(*
A circular queue implementation for managing `I_Arg`.  
*)
INTERFACE I_ArgQueue EXTENDS I_Debug

(*
Returns the current head index of the queue, indicating the next position for insertion.
*)
PROPERTY Head : UDINT
GET
END_GET
END_PROPERTY

PROPERTY Length : UDINT
GET
END_GET
END_PROPERTY

(*
Provides access to the underlying list structure that holds the queue's argument objects.
*)
PROPERTY List : I_ArgList
GET
END_GET
END_PROPERTY

(*
Returns the current tail index of the queue, indicating the next position for retrieval.
*)
PROPERTY Tail : UDINT
GET
END_GET
END_PROPERTY

END_INTERFACE

(* stored: Version 1.1.0.1
   Itf I_ArgQueue: Id {a3add385-e7ac-433c-818a-288d2bee859e}
   Property Head: Id {1e0693ff-f569-4e1a-858a-956b6e787fad}
   Get Get: Id {9e200817-2fc1-4cb6-b775-a63d6666a137}
   Property Length: Id {249cc34d-41f5-42c1-b7f3-69864b6b8d42}
   Get Get: Id {3e5ab514-7ad4-43a3-acb8-e66bc3d4d2ab}
   Property List: Id {ea10b641-3a44-49a3-8c2f-48f403aee4f0}
   Get Get: Id {1a2e15ab-7f7f-4c87-b178-b194d2df5ecc}
   Property Tail: Id {8b16c1d8-9ba4-45de-a37d-399410386f61}
   Get Get: Id {166a081e-a191-44c6-94eb-7586e93ce60b} *)
